PROGRAM Valvulas_Lavado
VAR
	ControlValv_ioLink_V6: ControlValv_ioLink;
	Falla_Lav_V6: BOOL;
	ControlValv_ioLink_V5: ControlValv_ioLink;
	Falla_Lav_V5: BOOL;
END_VAR
VAR // added by the converter: edge detectors and wires of the graphical bodies
    _w1, _w2 : BOOL;
END_VAR

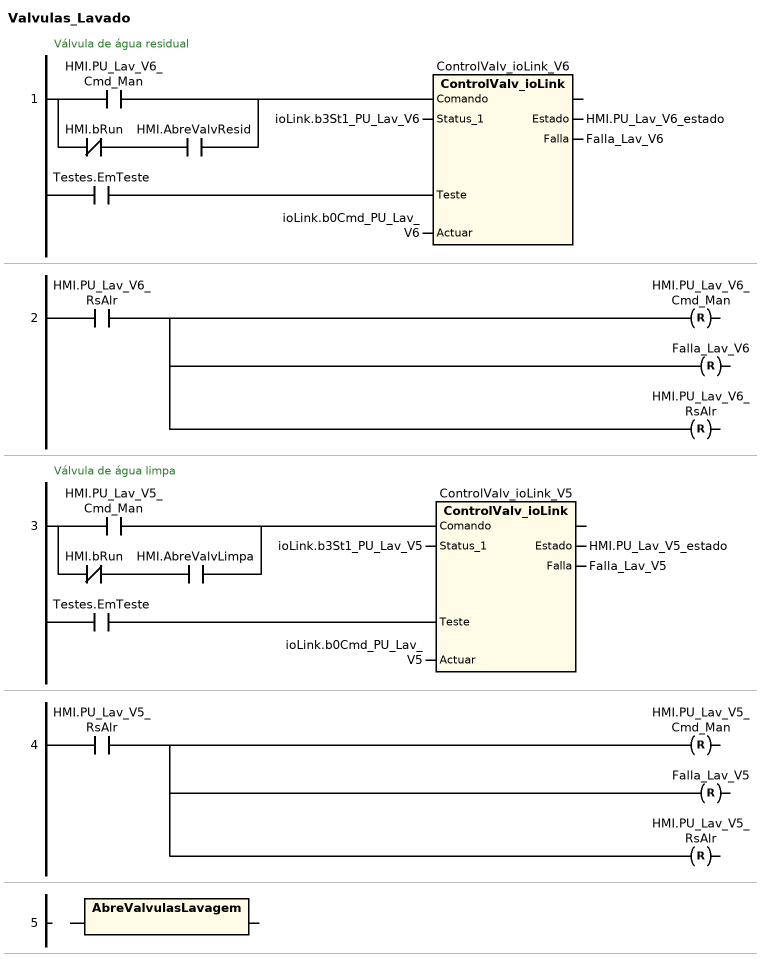
// NETWORK 1
// Válvula de água residual
ControlValv_ioLink_V6(
    Comando := HMI.PU_Lav_V6_Cmd_Man OR NOT HMI.bRun AND HMI.AbreValvResid,
    Status_1 := ioLink.b3St1_PU_Lav_V6,
    Teste := Testes.EmTeste,
    Actuar := ioLink.b0Cmd_PU_Lav_V6,
    Estado => HMI.PU_Lav_V6_estado,
    Falla => Falla_Lav_V6); // ControlValv_ioLink

// NETWORK 2
_w1 := HMI.PU_Lav_V6_RsAlr;
HMI.PU_Lav_V6_Cmd_Man R= _w1;
Falla_Lav_V6 R= _w1;
HMI.PU_Lav_V6_RsAlr R= _w1;

// NETWORK 3
// Válvula de água limpa
ControlValv_ioLink_V5(
    Comando := HMI.PU_Lav_V5_Cmd_Man OR NOT HMI.bRun AND HMI.AbreValvLimpa,
    Status_1 := ioLink.b3St1_PU_Lav_V5,
    Teste := Testes.EmTeste,
    Actuar := ioLink.b0Cmd_PU_Lav_V5,
    Estado => HMI.PU_Lav_V5_estado,
    Falla => Falla_Lav_V5); // ControlValv_ioLink

// NETWORK 4
_w2 := HMI.PU_Lav_V5_RsAlr;
HMI.PU_Lav_V5_Cmd_Man R= _w2;
Falla_Lav_V5 R= _w2;
HMI.PU_Lav_V5_RsAlr R= _w2;

// NETWORK 5
AbreValvulasLavagem();

END_PROGRAM

(* stored: Version 1.1.0.1, ProductVersion 3.1.4024.13
   POU Valvulas_Lavado: Id {6bb6d15c-d59b-4379-a87d-33b2a6586c35}, SpecialFunc None *)
